INTERFACE I_SignalHandling

METHOD Enable
VAR_INPUT
	bEnable		:		BOOL;
END_VAR
END_METHOD

METHOD SetOutput
VAR_INPUT
END_VAR
END_METHOD

END_INTERFACE

(* stored: Version 1.1.0.1, ProductVersion 3.1.4024.15
   Itf I_SignalHandling: Id {97ae229f-2e55-49a6-af87-27749c5819f6}
   Method Enable: Id {385c8dee-18f9-4cdd-85b3-ef3b0ac92ac8}
   Method SetOutput: Id {0bac8e01-62f1-4a95-9581-3b7c1410625e} *)
